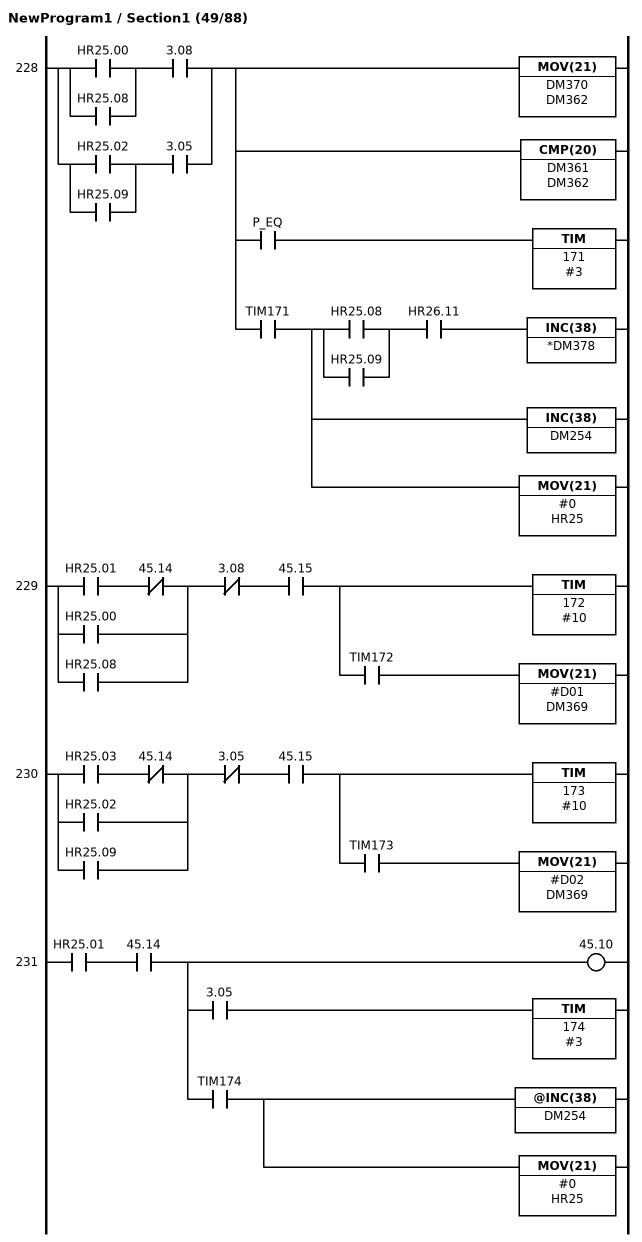
; [picture p48: NewProgram1 / Section1, rungs 228-231]
; rung 228
LD HR25.00
OR HR25.08
AND 3.08
LD HR25.02
OR HR25.09
AND 3.05
ORLD
OUT TR0
MOV(21) DM370 DM362
CMP(20) DM361 DM362
AND P_EQ
TIM 171 #3
LD TR0
AND TIM171
OUT TR0
LD HR25.08
OR HR25.09
ANDLD
AND HR26.11
INC(38) *DM378
LD TR0
INC(38) DM254
MOV(21) #0 HR25
; rung 229
LD HR25.01
ANDNOT 45.14
OR HR25.00
OR HR25.08
ANDNOT 3.08
AND 45.15
TIM 172 #10
AND TIM172
MOV(21) #D01 DM369
; rung 230
LD HR25.03
ANDNOT 45.14
OR HR25.02
OR HR25.09
ANDNOT 3.05
AND 45.15
TIM 173 #10
AND TIM173
MOV(21) #D02 DM369
; rung 231
LD HR25.01
AND 45.14
OUT TR0
OUT 45.10
AND 3.05
TIM 174 #3
LD TR0
AND TIM174
@INC(38) DM254
MOV(21) #0 HR25

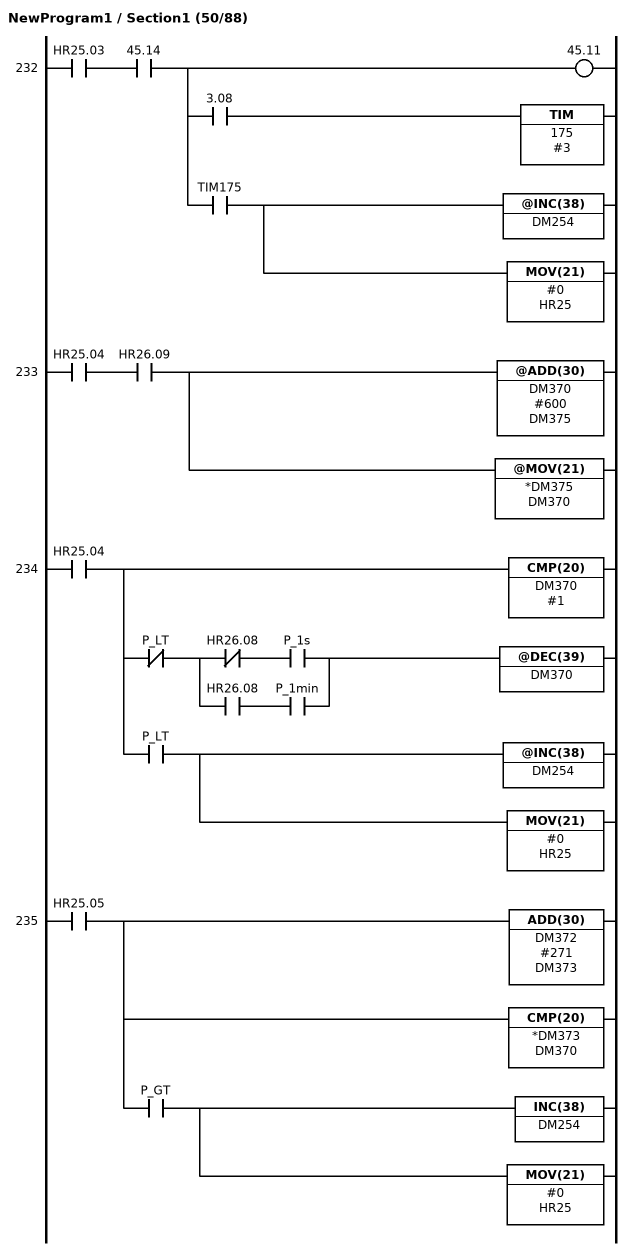
; rung 232
LD HR25.03
AND 45.14
OUT TR0
OUT 45.11
AND 3.08
TIM 175 #3
LD TR0
AND TIM175
@INC(38) DM254
MOV(21) #0 HR25
; rung 233
LD HR25.04
AND HR26.09
@ADD(30) DM370 #600 DM375
@MOV(21) *DM375 DM370
; rung 234
LD HR25.04
OUT TR0
CMP(20) DM370 #1
ANDNOT P_LT
LDNOT HR26.08
AND P_1s
LD HR26.08
AND P_1min
ORLD
ANDLD
@DEC(39) DM370
LD TR0
AND P_LT
@INC(38) DM254
MOV(21) #0 HR25
; rung 235
LD HR25.05
ADD(30) DM372 #271 DM373
CMP(20) *DM373 DM370
AND P_GT
INC(38) DM254
MOV(21) #0 HR25

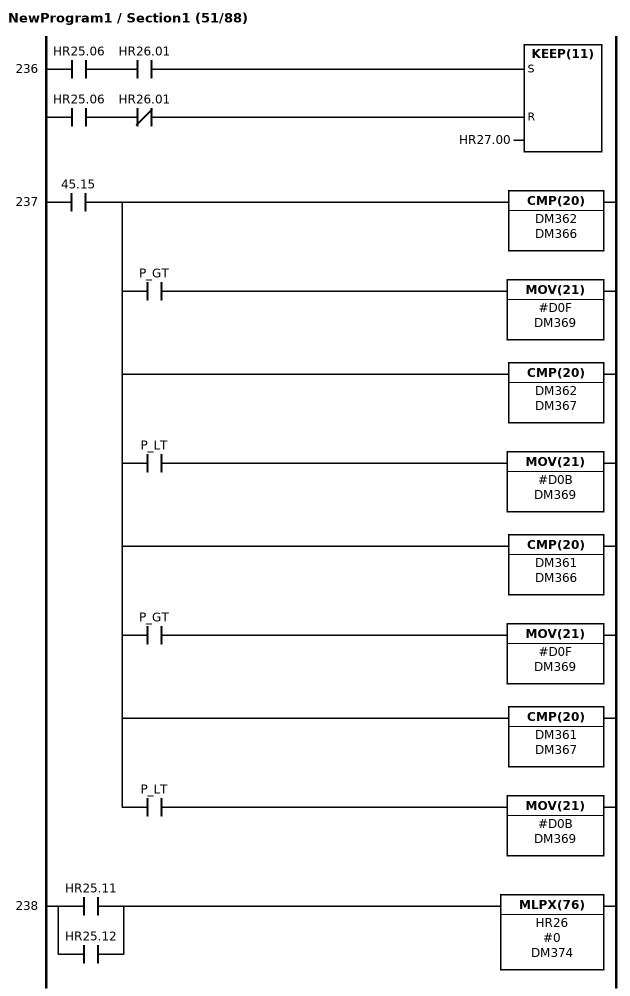
; rung 236
LD HR25.06
AND HR26.01
LD HR25.06
ANDNOT HR26.01
KEEP(11) HR27.00
; rung 237
LD 45.15
OUT TR0
CMP(20) DM362 DM366
AND P_GT
MOV(21) #D0F DM369
LD TR0
CMP(20) DM362 DM367
AND P_LT
MOV(21) #D0B DM369
LD TR0
CMP(20) DM361 DM366
AND P_GT
MOV(21) #D0F DM369
LD TR0
CMP(20) DM361 DM367
AND P_LT
MOV(21) #D0B DM369
; rung 238
LD HR25.11
OR HR25.12
MLPX(76) HR26 #0 DM374

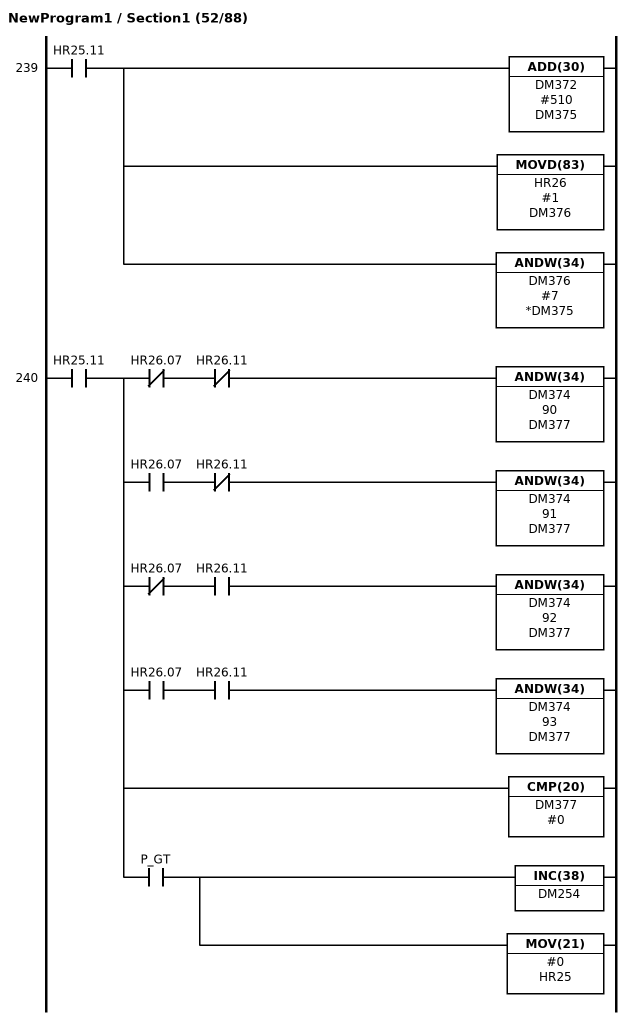
; rung 239
LD HR25.11
ADD(30) DM372 #510 DM375
MOVD(83) HR26 #1 DM376
ANDW(34) DM376 #7 *DM375
; rung 240
LD HR25.11
OUT TR0
ANDNOT HR26.07
ANDNOT HR26.11
ANDW(34) DM374 90 DM377
LD TR0
AND HR26.07
ANDNOT HR26.11
ANDW(34) DM374 91 DM377
LD TR0
ANDNOT HR26.07
AND HR26.11
ANDW(34) DM374 92 DM377
LD TR0
AND HR26.07
AND HR26.11
ANDW(34) DM374 93 DM377
LD TR0
CMP(20) DM377 #0
AND P_GT
INC(38) DM254
MOV(21) #0 HR25

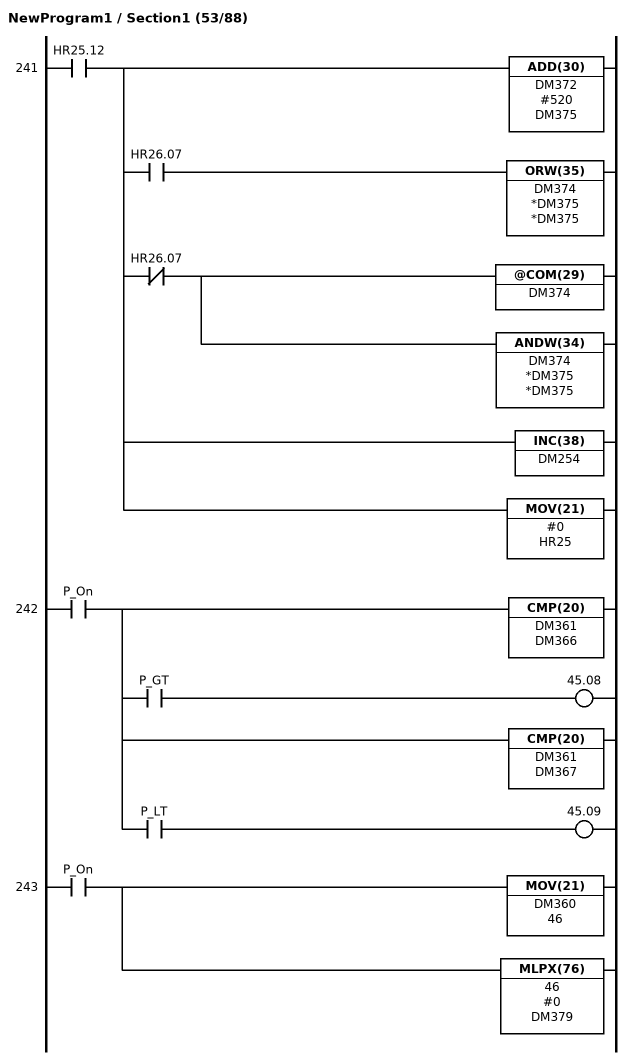
; rung 241
LD HR25.12
OUT TR0
ADD(30) DM372 #520 DM375
AND HR26.07
ORW(35) DM374 *DM375 *DM375
LD TR0
ANDNOT HR26.07
@COM(29) DM374
ANDW(34) DM374 *DM375 *DM375
LD TR0
INC(38) DM254
MOV(21) #0 HR25
; rung 242
LD P_On
OUT TR0
CMP(20) DM361 DM366
AND P_GT
OUT 45.08
LD TR0
CMP(20) DM361 DM367
AND P_LT
OUT 45.09
; rung 243
LD P_On
MOV(21) DM360 46
MLPX(76) 46 #0 DM379

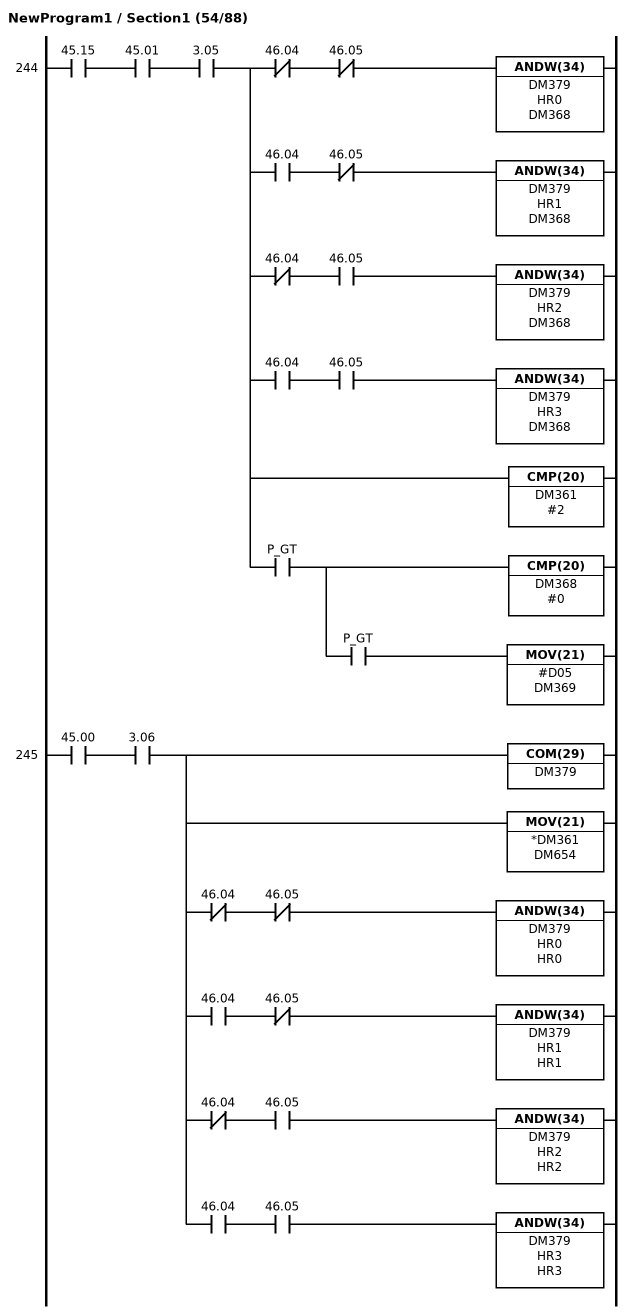
; rung 244
LD 45.15
AND 45.01
AND 3.05
OUT TR0
ANDNOT 46.04
ANDNOT 46.05
ANDW(34) DM379 HR0 DM368
LD TR0
AND 46.04
ANDNOT 46.05
ANDW(34) DM379 HR1 DM368
LD TR0
ANDNOT 46.04
AND 46.05
ANDW(34) DM379 HR2 DM368
LD TR0
AND 46.04
AND 46.05
ANDW(34) DM379 HR3 DM368
LD TR0
CMP(20) DM361 #2
AND P_GT
CMP(20) DM368 #0
AND P_GT
MOV(21) #D05 DM369
; rung 245
LD 45.00
AND 3.06
OUT TR0
COM(29) DM379
MOV(21) *DM361 DM654
ANDNOT 46.04
ANDNOT 46.05
ANDW(34) DM379 HR0 HR0
LD TR0
AND 46.04
ANDNOT 46.05
ANDW(34) DM379 HR1 HR1
LD TR0
ANDNOT 46.04
AND 46.05
ANDW(34) DM379 HR2 HR2
LD TR0
AND 46.04
AND 46.05
ANDW(34) DM379 HR3 HR3

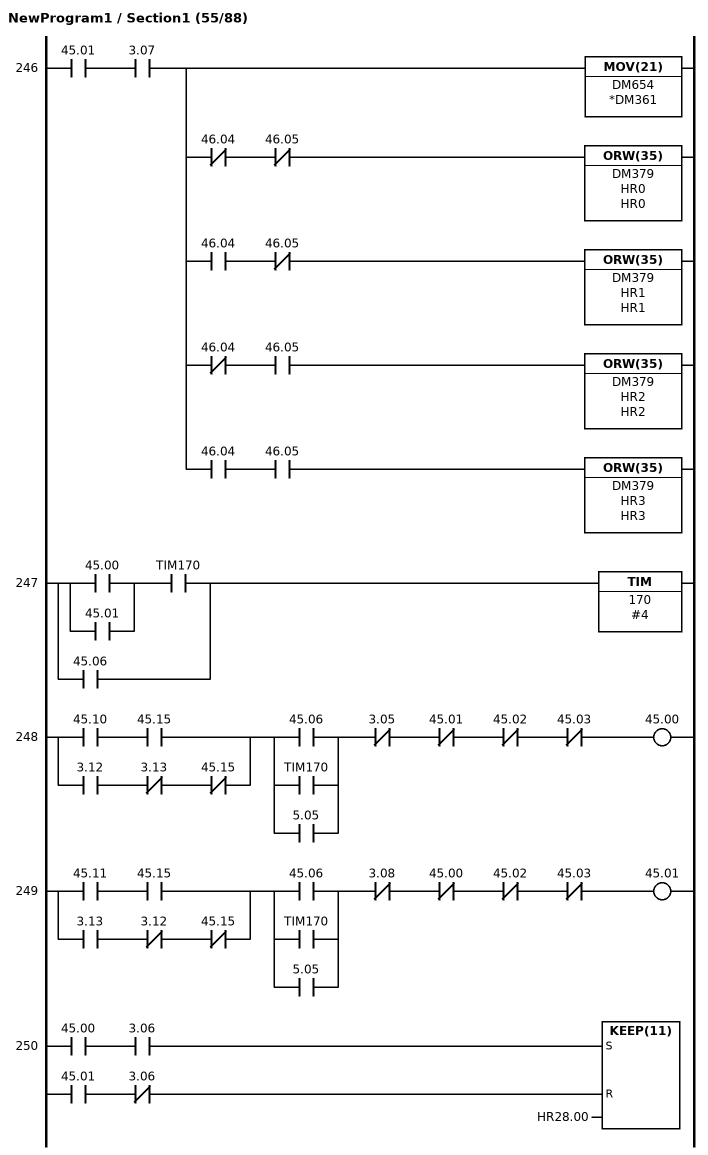
; rung 246
LD 45.01
AND 3.07
OUT TR0
MOV(21) DM654 *DM361
ANDNOT 46.04
ANDNOT 46.05
ORW(35) DM379 HR0 HR0
LD TR0
AND 46.04
ANDNOT 46.05
ORW(35) DM379 HR1 HR1
LD TR0
ANDNOT 46.04
AND 46.05
ORW(35) DM379 HR2 HR2
LD TR0
AND 46.04
AND 46.05
ORW(35) DM379 HR3 HR3
; rung 247
LD 45.00
OR 45.01
AND TIM170
OR 45.06
TIM 170 #4
; rung 248
LD 45.10
AND 45.15
LD 3.12
ANDNOT 3.13
ANDNOT 45.15
ORLD
LD 45.06
OR TIM170
OR 5.05
ANDLD
ANDNOT 3.05
ANDNOT 45.01
ANDNOT 45.02
ANDNOT 45.03
OUT 45.00
; rung 249
LD 45.11
AND 45.15
LD 3.13
ANDNOT 3.12
ANDNOT 45.15
ORLD
LD 45.06
OR TIM170
OR 5.05
ANDLD
ANDNOT 3.08
ANDNOT 45.00
ANDNOT 45.02
ANDNOT 45.03
OUT 45.01
; rung 250
LD 45.00
AND 3.06
LD 45.01
ANDNOT 3.06
KEEP(11) HR28.00

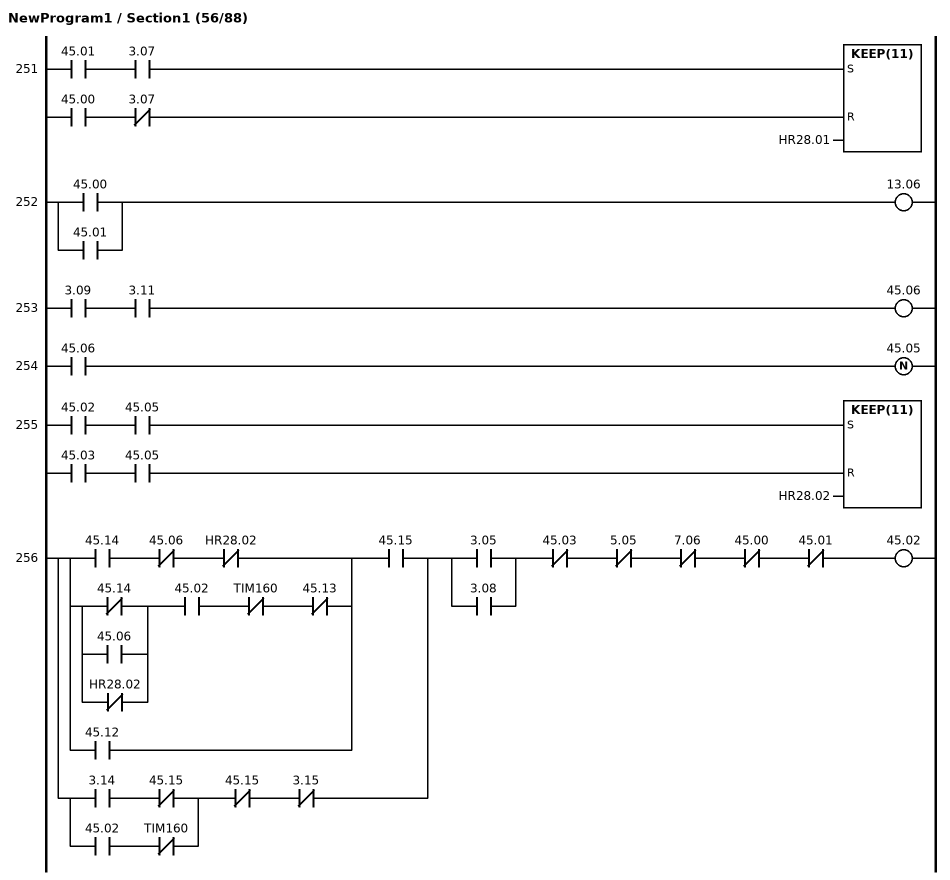
; rung 251
LD 45.01
AND 3.07
LD 45.00
ANDNOT 3.07
KEEP(11) HR28.01
; rung 252
LD 45.00
OR 45.01
OUT 13.06
; rung 253
LD 3.09
AND 3.11
OUT 45.06
; rung 254
LD 45.06
DIFD(14) 45.05
; rung 255
LD 45.02
AND 45.05
LD 45.03
AND 45.05
KEEP(11) HR28.02
; rung 256
LD 45.14
ANDNOT 45.06
ANDNOT HR28.02
LDNOT 45.14
OR 45.06
ORNOT HR28.02
AND 45.02
ANDNOT TIM160
ANDNOT 45.13
ORLD
OR 45.12
AND 45.15
LD 3.14
ANDNOT 45.15
LD 45.02
ANDNOT TIM160
ORLD
ANDNOT 45.15
ANDNOT 3.15
ORLD
LD 3.05
OR 3.08
ANDLD
ANDNOT 45.03
ANDNOT 5.05
ANDNOT 7.06
ANDNOT 45.00
ANDNOT 45.01
OUT 45.02

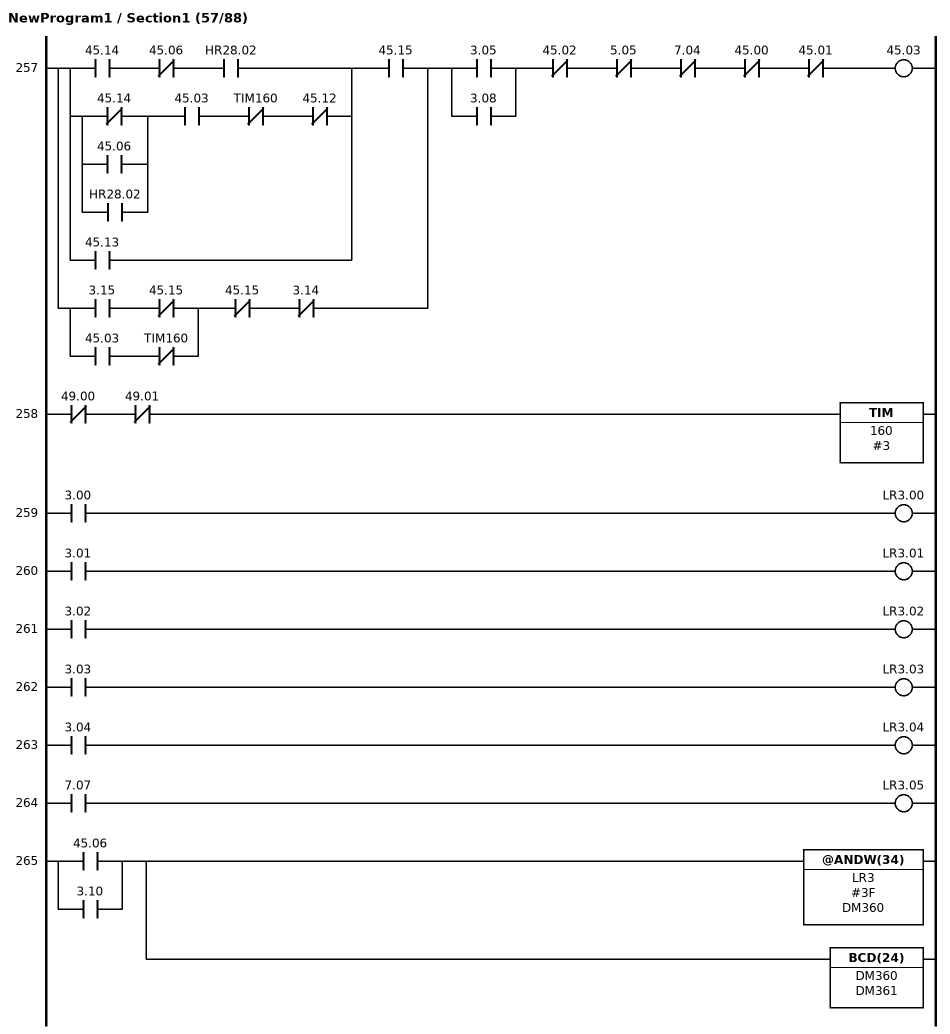
; rung 257
LD 45.14
ANDNOT 45.06
AND HR28.02
LDNOT 45.14
OR 45.06
OR HR28.02
AND 45.03
ANDNOT TIM160
ANDNOT 45.12
ORLD
OR 45.13
AND 45.15
LD 3.15
ANDNOT 45.15
LD 45.03
ANDNOT TIM160
ORLD
ANDNOT 45.15
ANDNOT 3.14
ORLD
LD 3.05
OR 3.08
ANDLD
ANDNOT 45.02
ANDNOT 5.05
ANDNOT 7.04
ANDNOT 45.00
ANDNOT 45.01
OUT 45.03
; rung 258
LDNOT 49.00
ANDNOT 49.01
TIM 160 #3
; rung 259
LD 3.00
OUT LR3.00
; rung 260
LD 3.01
OUT LR3.01
; rung 261
LD 3.02
OUT LR3.02
; rung 262
LD 3.03
OUT LR3.03
; rung 263
LD 3.04
OUT LR3.04
; rung 264
LD 7.07
OUT LR3.05
; rung 265
LD 45.06
OR 3.10
@ANDW(34) LR3 #3F DM360
BCD(24) DM360 DM361

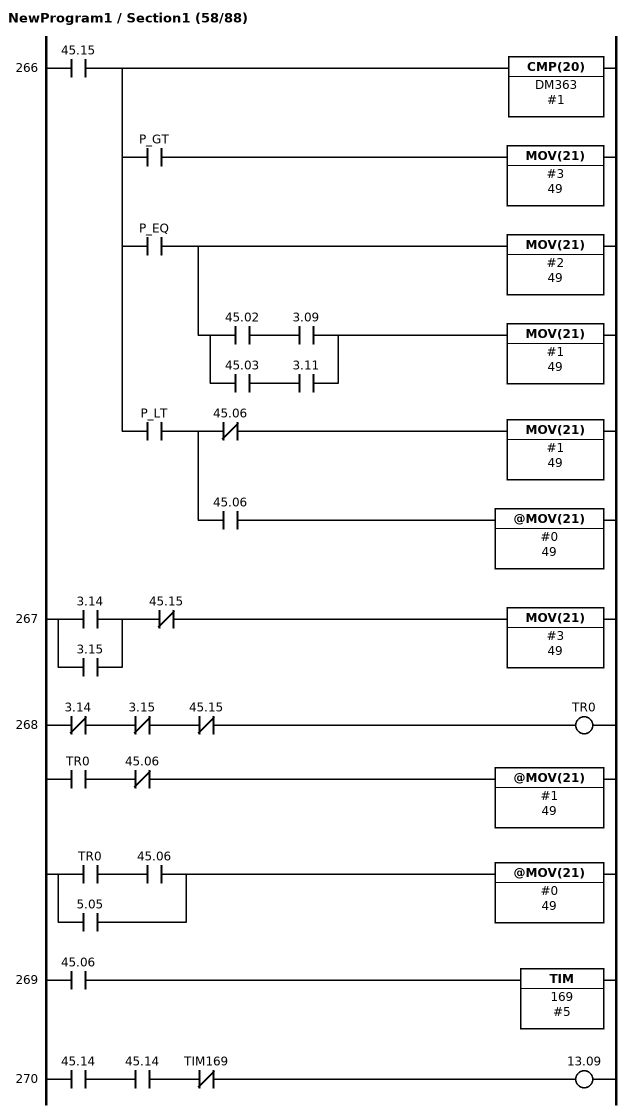
; rung 266
LD 45.15
OUT TR0
CMP(20) DM363 #1
AND P_GT
MOV(21) #3 49
LD TR0
AND P_EQ
MOV(21) #2 49
LD 45.02
AND 3.09
LD 45.03
AND 3.11
ORLD
ANDLD
MOV(21) #1 49
LD TR0
AND P_LT
OUT TR0
ANDNOT 45.06
MOV(21) #1 49
LD TR0
AND 45.06
@MOV(21) #0 49
; rung 267
LD 3.14
OR 3.15
ANDNOT 45.15
MOV(21) #3 49
; rung 268
LDNOT 3.14
ANDNOT 3.15
ANDNOT 45.15
OUT TR0
ANDNOT 45.06
@MOV(21) #1 49
LD TR0
AND 45.06
OR 5.05
@MOV(21) #0 49
; rung 269
LD 45.06
TIM 169 #5
; rung 270
LD 45.14
AND 45.14
ANDNOT TIM169
OUT 13.09

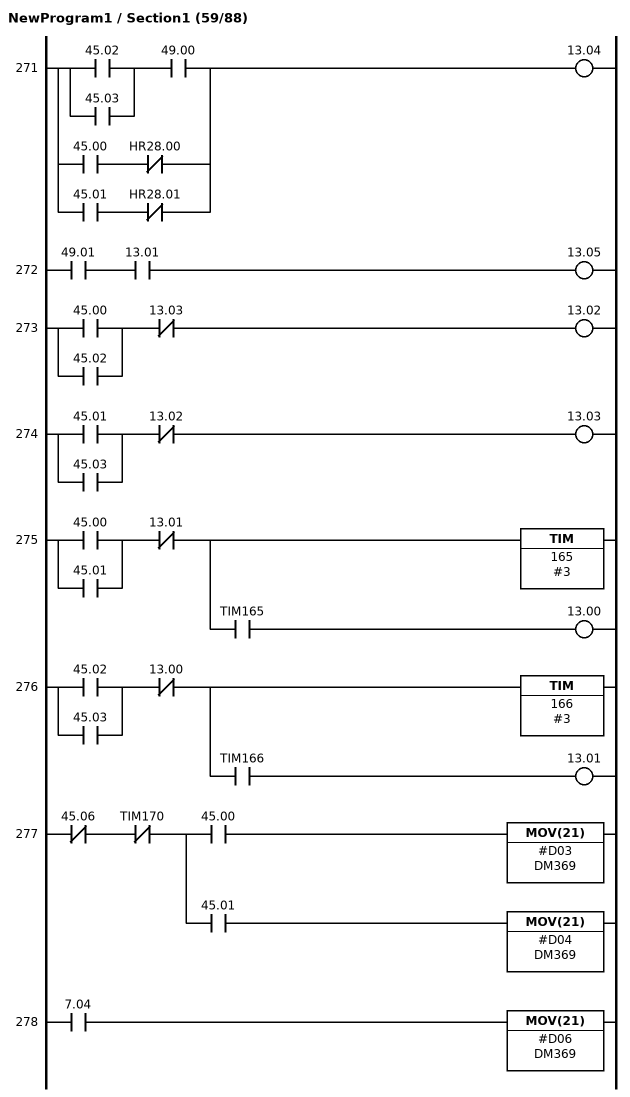
; rung 271
LD 45.02
OR 45.03
AND 49.00
LD 45.00
ANDNOT HR28.00
ORLD
LD 45.01
ANDNOT HR28.01
ORLD
OUT 13.04
; rung 272
LD 49.01
AND 13.01
OUT 13.05
; rung 273
LD 45.00
OR 45.02
ANDNOT 13.03
OUT 13.02
; rung 274
LD 45.01
OR 45.03
ANDNOT 13.02
OUT 13.03
; rung 275
LD 45.00
OR 45.01
ANDNOT 13.01
TIM 165 #3
AND TIM165
OUT 13.00
; rung 276
LD 45.02
OR 45.03
ANDNOT 13.00
TIM 166 #3
AND TIM166
OUT 13.01
; rung 277
LDNOT 45.06
ANDNOT TIM170
OUT TR0
AND 45.00
MOV(21) #D03 DM369
LD TR0
AND 45.01
MOV(21) #D04 DM369
; rung 278
LD 7.04
MOV(21) #D06 DM369

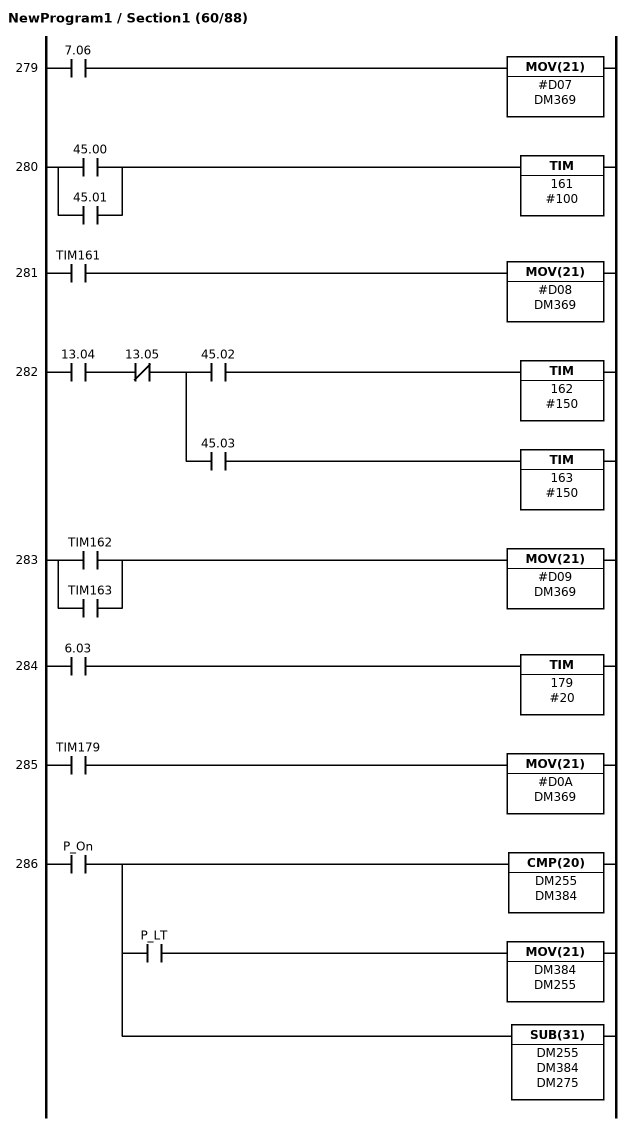
; rung 279
LD 7.06
MOV(21) #D07 DM369
; rung 280
LD 45.00
OR 45.01
TIM 161 #100
; rung 281
LD TIM161
MOV(21) #D08 DM369
; rung 282
LD 13.04
ANDNOT 13.05
OUT TR0
AND 45.02
TIM 162 #150
LD TR0
AND 45.03
TIM 163 #150
; rung 283
LD TIM162
OR TIM163
MOV(21) #D09 DM369
; rung 284
LD 6.03
TIM 179 #20
; rung 285
LD TIM179
MOV(21) #D0A DM369
; rung 286
LD P_On
OUT TR0
CMP(20) DM255 DM384
AND P_LT
MOV(21) DM384 DM255
LD TR0
SUB(31) DM255 DM384 DM275

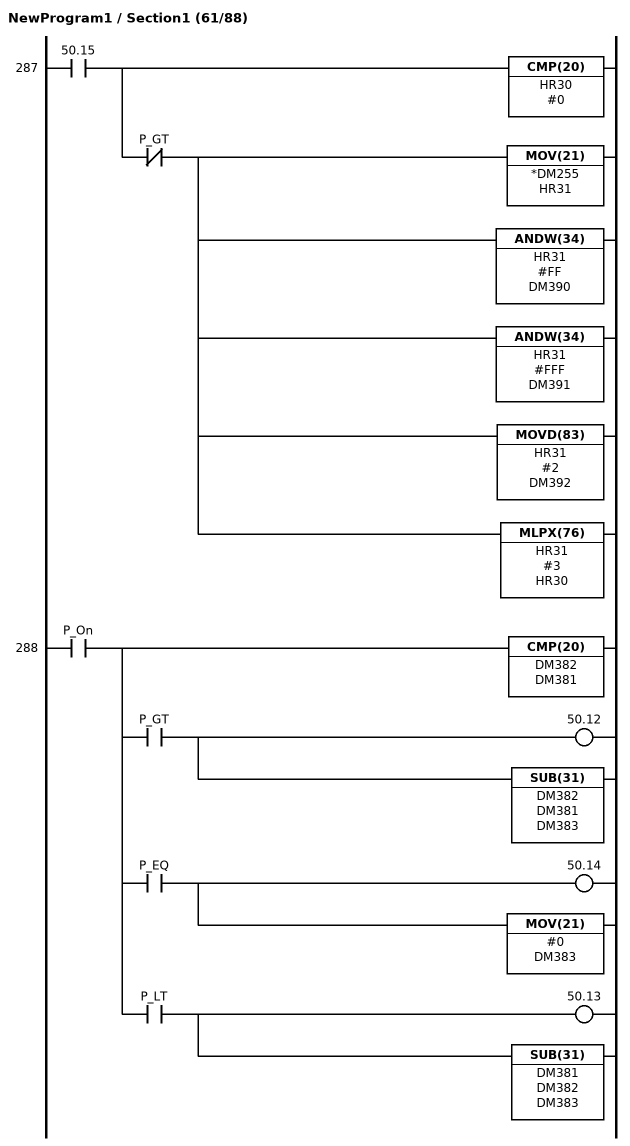
; rung 287
LD 50.15
CMP(20) HR30 #0
ANDNOT P_GT
MOV(21) *DM255 HR31
ANDW(34) HR31 #FF DM390
ANDW(34) HR31 #FFF DM391
MOVD(83) HR31 #2 DM392
MLPX(76) HR31 #3 HR30
; rung 288
LD P_On
OUT TR0
CMP(20) DM382 DM381
AND P_GT
OUT 50.12
SUB(31) DM382 DM381 DM383
LD TR0
AND P_EQ
OUT 50.14
MOV(21) #0 DM383
LD TR0
AND P_LT
OUT 50.13
SUB(31) DM381 DM382 DM383

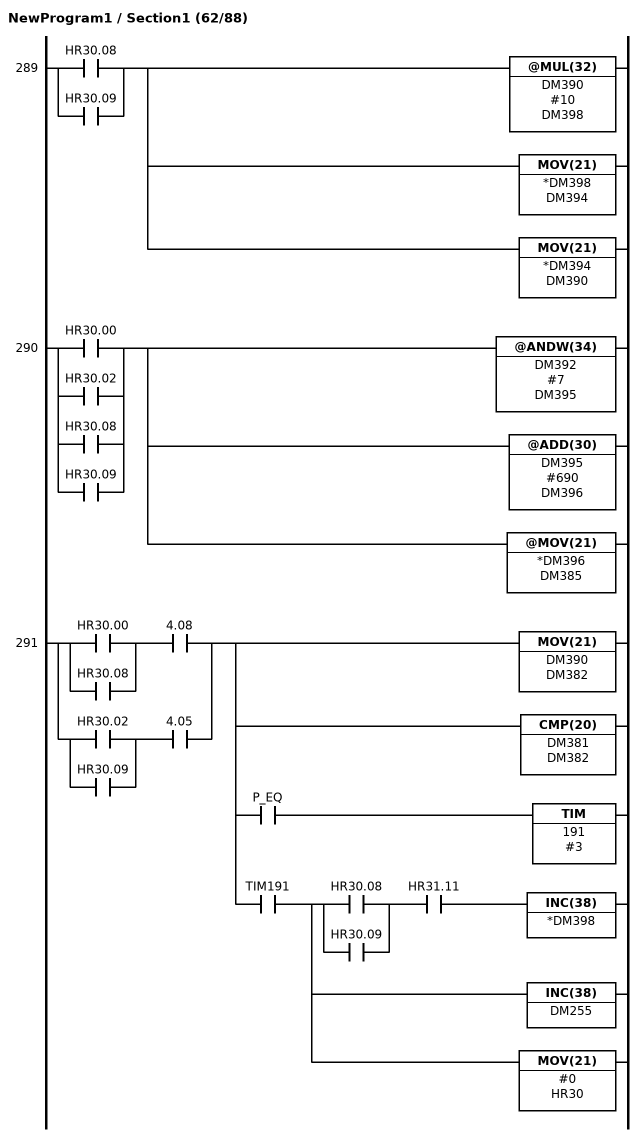
; rung 289
LD HR30.08
OR HR30.09
@MUL(32) DM390 #10 DM398
MOV(21) *DM398 DM394
MOV(21) *DM394 DM390
; rung 290
LD HR30.00
OR HR30.02
OR HR30.08
OR HR30.09
@ANDW(34) DM392 #7 DM395
@ADD(30) DM395 #690 DM396
@MOV(21) *DM396 DM385
; rung 291
LD HR30.00
OR HR30.08
AND 4.08
LD HR30.02
OR HR30.09
AND 4.05
ORLD
OUT TR0
MOV(21) DM390 DM382
CMP(20) DM381 DM382
AND P_EQ
TIM 191 #3
LD TR0
AND TIM191
OUT TR0
LD HR30.08
OR HR30.09
ANDLD
AND HR31.11
INC(38) *DM398
LD TR0
INC(38) DM255
MOV(21) #0 HR30

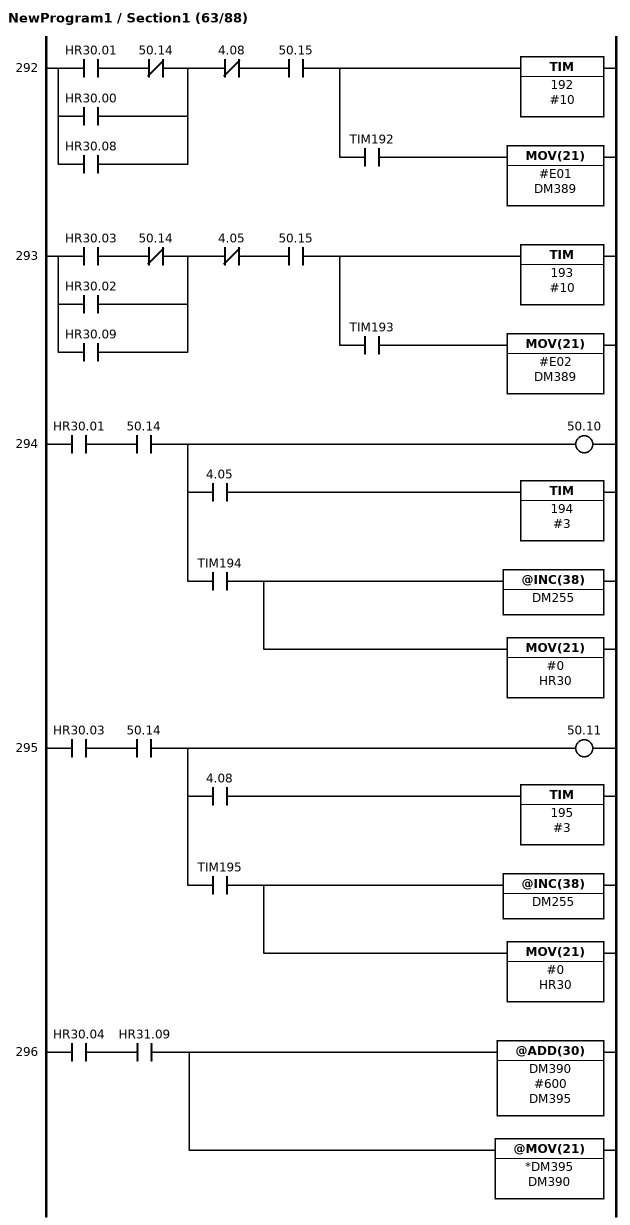
; rung 292
LD HR30.01
ANDNOT 50.14
OR HR30.00
OR HR30.08
ANDNOT 4.08
AND 50.15
TIM 192 #10
AND TIM192
MOV(21) #E01 DM389
; rung 293
LD HR30.03
ANDNOT 50.14
OR HR30.02
OR HR30.09
ANDNOT 4.05
AND 50.15
TIM 193 #10
AND TIM193
MOV(21) #E02 DM389
; rung 294
LD HR30.01
AND 50.14
OUT TR0
OUT 50.10
AND 4.05
TIM 194 #3
LD TR0
AND TIM194
@INC(38) DM255
MOV(21) #0 HR30
; rung 295
LD HR30.03
AND 50.14
OUT TR0
OUT 50.11
AND 4.08
TIM 195 #3
LD TR0
AND TIM195
@INC(38) DM255
MOV(21) #0 HR30
; rung 296
LD HR30.04
AND HR31.09
@ADD(30) DM390 #600 DM395
@MOV(21) *DM395 DM390

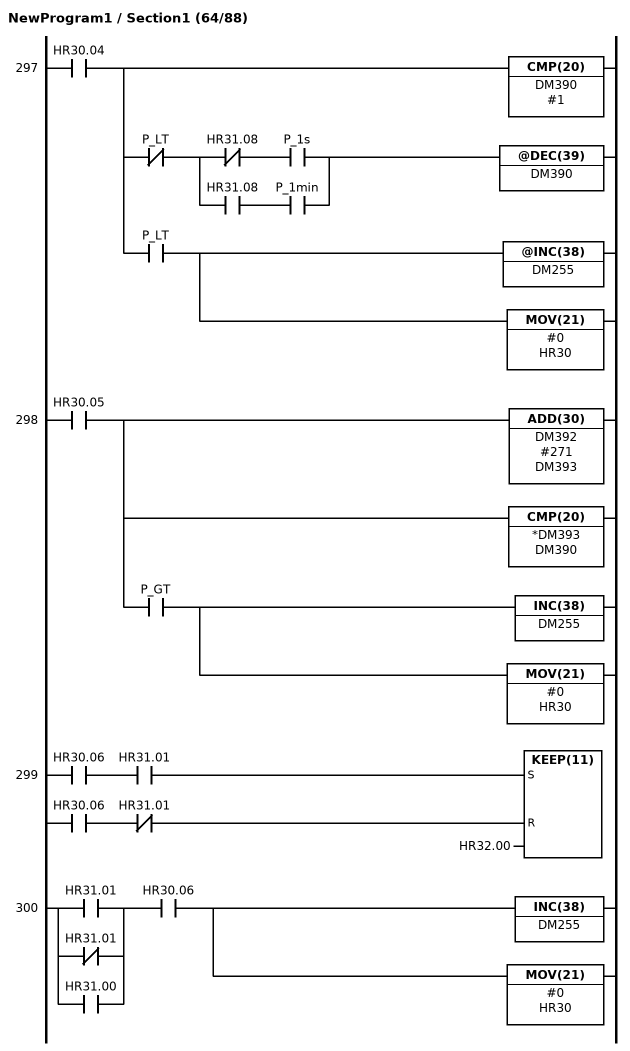
; rung 297
LD HR30.04
OUT TR0
CMP(20) DM390 #1
ANDNOT P_LT
LDNOT HR31.08
AND P_1s
LD HR31.08
AND P_1min
ORLD
ANDLD
@DEC(39) DM390
LD TR0
AND P_LT
@INC(38) DM255
MOV(21) #0 HR30
; rung 298
LD HR30.05
ADD(30) DM392 #271 DM393
CMP(20) *DM393 DM390
AND P_GT
INC(38) DM255
MOV(21) #0 HR30
; rung 299
LD HR30.06
AND HR31.01
LD HR30.06
ANDNOT HR31.01
KEEP(11) HR32.00
; rung 300
LD HR31.01
ORNOT HR31.01
OR HR31.00
AND HR30.06
INC(38) DM255
MOV(21) #0 HR30

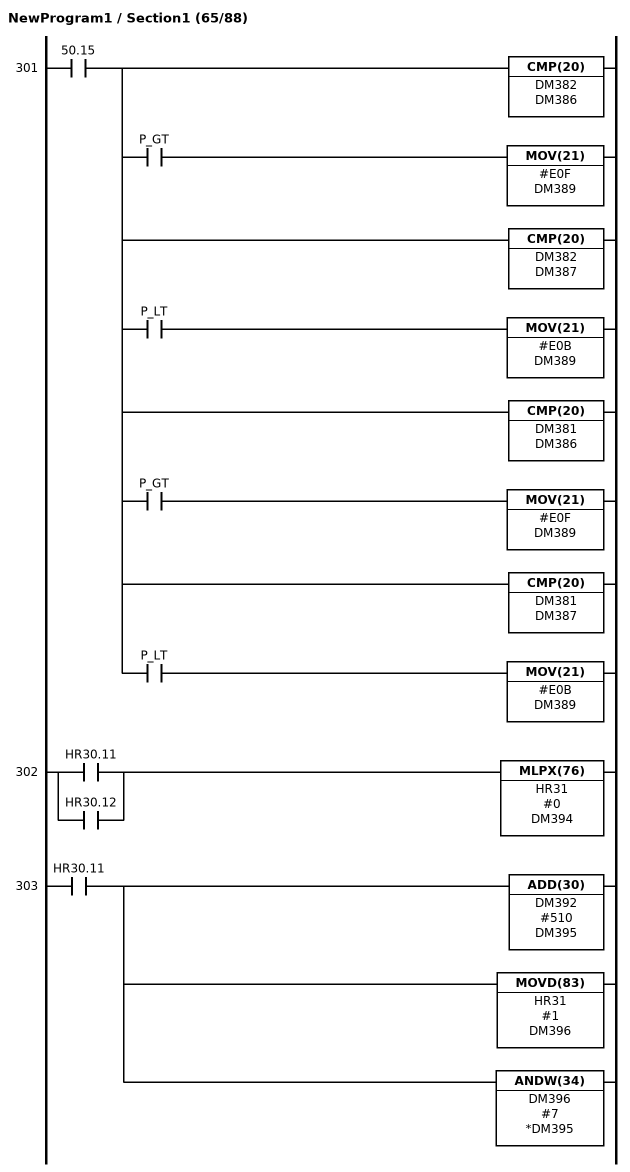
; rung 301
LD 50.15
OUT TR0
CMP(20) DM382 DM386
AND P_GT
MOV(21) #E0F DM389
LD TR0
CMP(20) DM382 DM387
AND P_LT
MOV(21) #E0B DM389
LD TR0
CMP(20) DM381 DM386
AND P_GT
MOV(21) #E0F DM389
LD TR0
CMP(20) DM381 DM387
AND P_LT
MOV(21) #E0B DM389
; rung 302
LD HR30.11
OR HR30.12
MLPX(76) HR31 #0 DM394
; rung 303
LD HR30.11
ADD(30) DM392 #510 DM395
MOVD(83) HR31 #1 DM396
ANDW(34) DM396 #7 *DM395

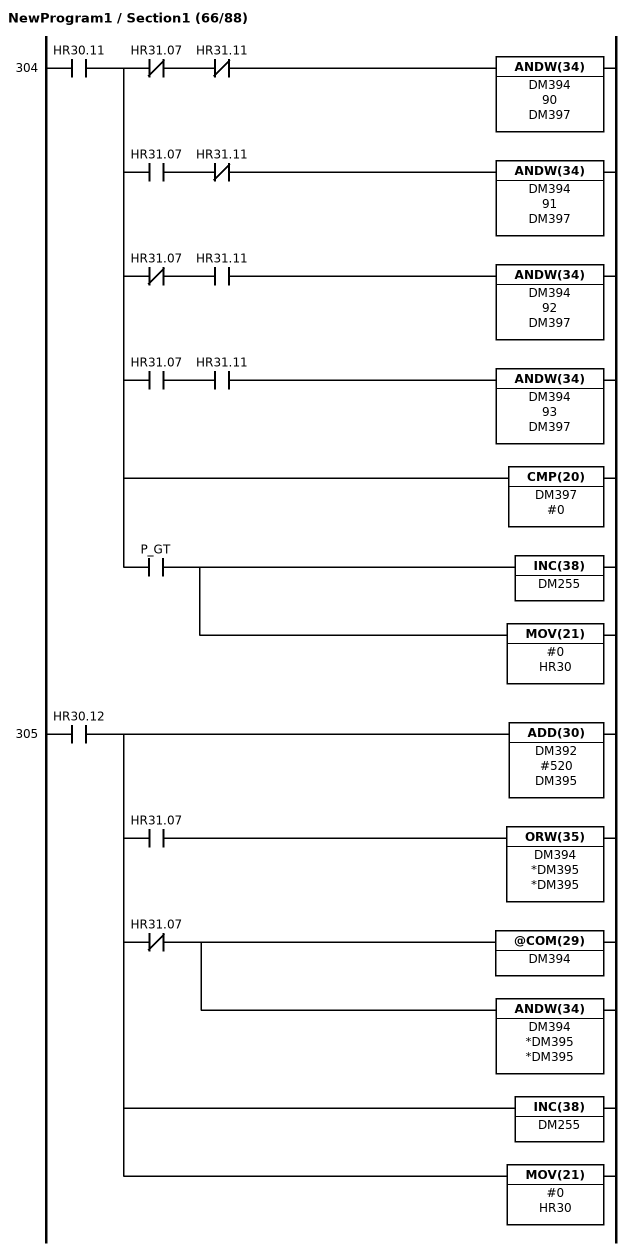
; rung 304
LD HR30.11
OUT TR0
ANDNOT HR31.07
ANDNOT HR31.11
ANDW(34) DM394 90 DM397
LD TR0
AND HR31.07
ANDNOT HR31.11
ANDW(34) DM394 91 DM397
LD TR0
ANDNOT HR31.07
AND HR31.11
ANDW(34) DM394 92 DM397
LD TR0
AND HR31.07
AND HR31.11
ANDW(34) DM394 93 DM397
LD TR0
CMP(20) DM397 #0
AND P_GT
INC(38) DM255
MOV(21) #0 HR30
; rung 305
LD HR30.12
OUT TR0
ADD(30) DM392 #520 DM395
AND HR31.07
ORW(35) DM394 *DM395 *DM395
LD TR0
ANDNOT HR31.07
@COM(29) DM394
ANDW(34) DM394 *DM395 *DM395
LD TR0
INC(38) DM255
MOV(21) #0 HR30

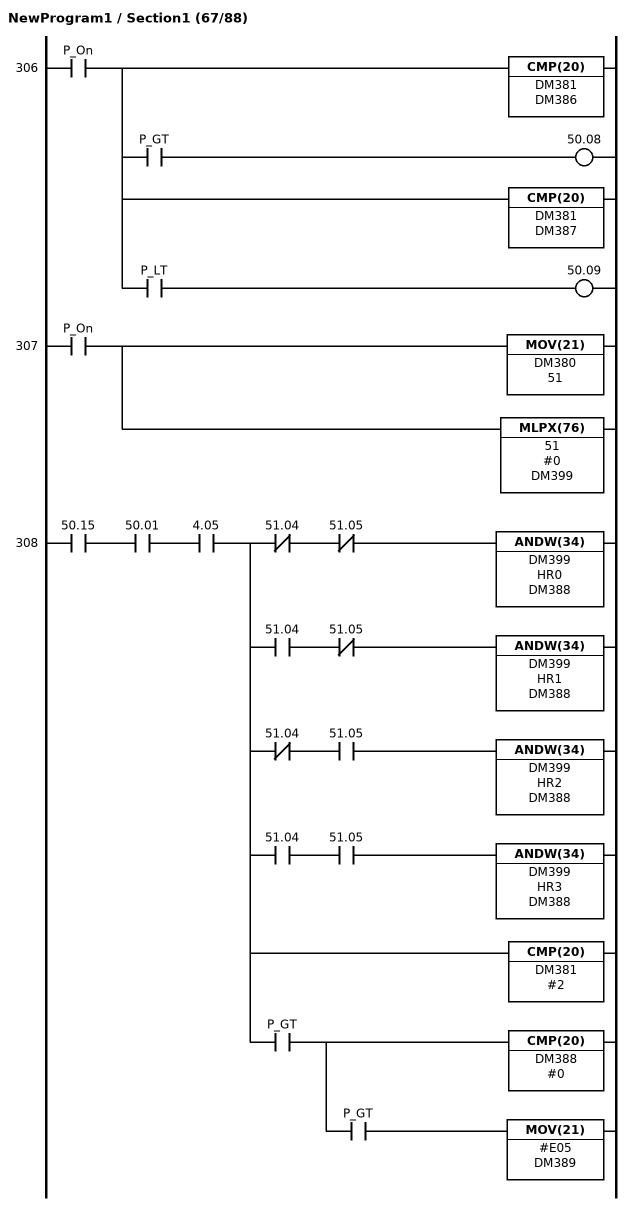
; rung 306
LD P_On
OUT TR0
CMP(20) DM381 DM386
AND P_GT
OUT 50.08
LD TR0
CMP(20) DM381 DM387
AND P_LT
OUT 50.09
; rung 307
LD P_On
MOV(21) DM380 51
MLPX(76) 51 #0 DM399
; rung 308
LD 50.15
AND 50.01
AND 4.05
OUT TR0
ANDNOT 51.04
ANDNOT 51.05
ANDW(34) DM399 HR0 DM388
LD TR0
AND 51.04
ANDNOT 51.05
ANDW(34) DM399 HR1 DM388
LD TR0
ANDNOT 51.04
AND 51.05
ANDW(34) DM399 HR2 DM388
LD TR0
AND 51.04
AND 51.05
ANDW(34) DM399 HR3 DM388
LD TR0
CMP(20) DM381 #2
AND P_GT
CMP(20) DM388 #0
AND P_GT
MOV(21) #E05 DM389

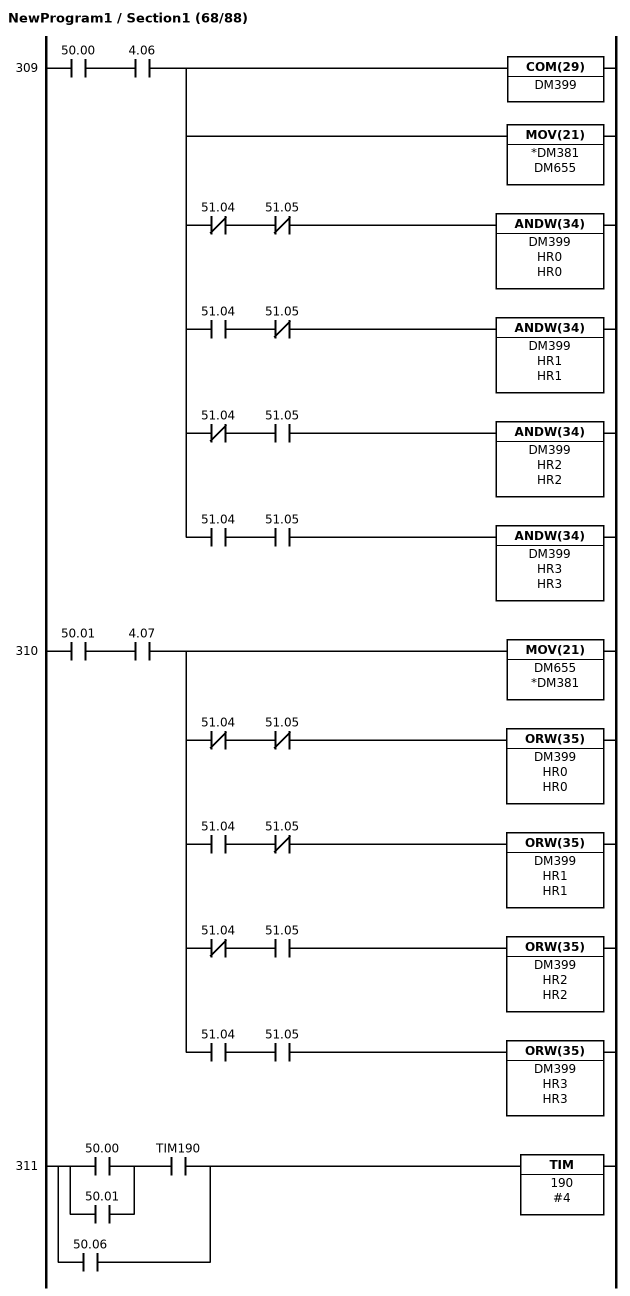
; rung 309
LD 50.00
AND 4.06
OUT TR0
COM(29) DM399
MOV(21) *DM381 DM655
ANDNOT 51.04
ANDNOT 51.05
ANDW(34) DM399 HR0 HR0
LD TR0
AND 51.04
ANDNOT 51.05
ANDW(34) DM399 HR1 HR1
LD TR0
ANDNOT 51.04
AND 51.05
ANDW(34) DM399 HR2 HR2
LD TR0
AND 51.04
AND 51.05
ANDW(34) DM399 HR3 HR3
; rung 310
LD 50.01
AND 4.07
OUT TR0
MOV(21) DM655 *DM381
ANDNOT 51.04
ANDNOT 51.05
ORW(35) DM399 HR0 HR0
LD TR0
AND 51.04
ANDNOT 51.05
ORW(35) DM399 HR1 HR1
LD TR0
ANDNOT 51.04
AND 51.05
ORW(35) DM399 HR2 HR2
LD TR0
AND 51.04
AND 51.05
ORW(35) DM399 HR3 HR3
; rung 311
LD 50.00
OR 50.01
AND TIM190
OR 50.06
TIM 190 #4

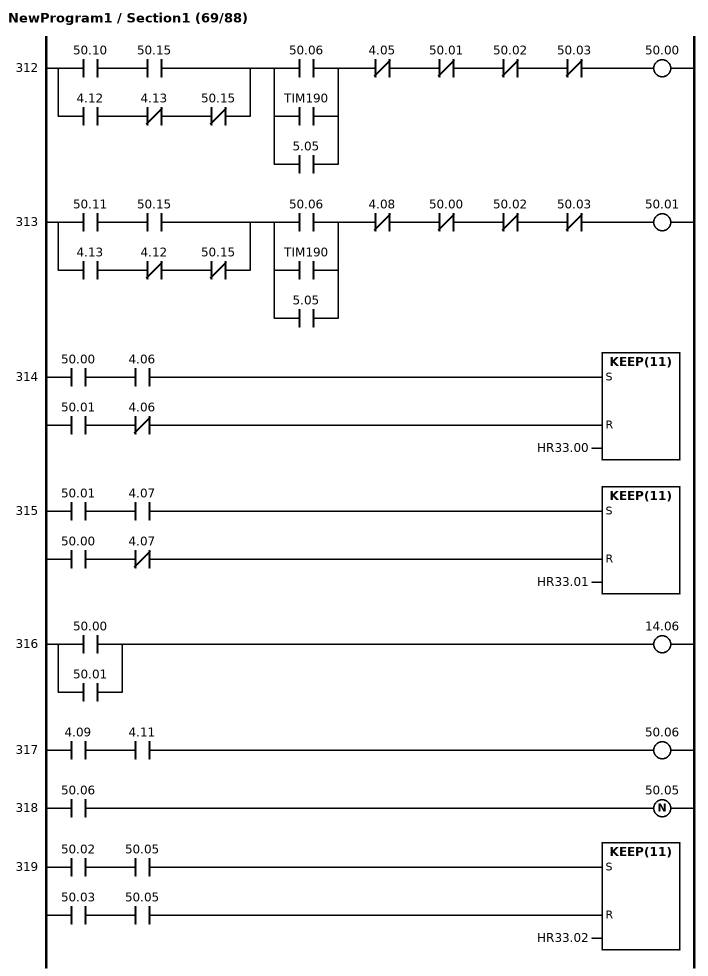
; rung 312
LD 50.10
AND 50.15
LD 4.12
ANDNOT 4.13
ANDNOT 50.15
ORLD
LD 50.06
OR TIM190
OR 5.05
ANDLD
ANDNOT 4.05
ANDNOT 50.01
ANDNOT 50.02
ANDNOT 50.03
OUT 50.00
; rung 313
LD 50.11
AND 50.15
LD 4.13
ANDNOT 4.12
ANDNOT 50.15
ORLD
LD 50.06
OR TIM190
OR 5.05
ANDLD
ANDNOT 4.08
ANDNOT 50.00
ANDNOT 50.02
ANDNOT 50.03
OUT 50.01
; rung 314
LD 50.00
AND 4.06
LD 50.01
ANDNOT 4.06
KEEP(11) HR33.00
; rung 315
LD 50.01
AND 4.07
LD 50.00
ANDNOT 4.07
KEEP(11) HR33.01
; rung 316
LD 50.00
OR 50.01
OUT 14.06
; rung 317
LD 4.09
AND 4.11
OUT 50.06
; rung 318
LD 50.06
DIFD(14) 50.05
; rung 319
LD 50.02
AND 50.05
LD 50.03
AND 50.05
KEEP(11) HR33.02

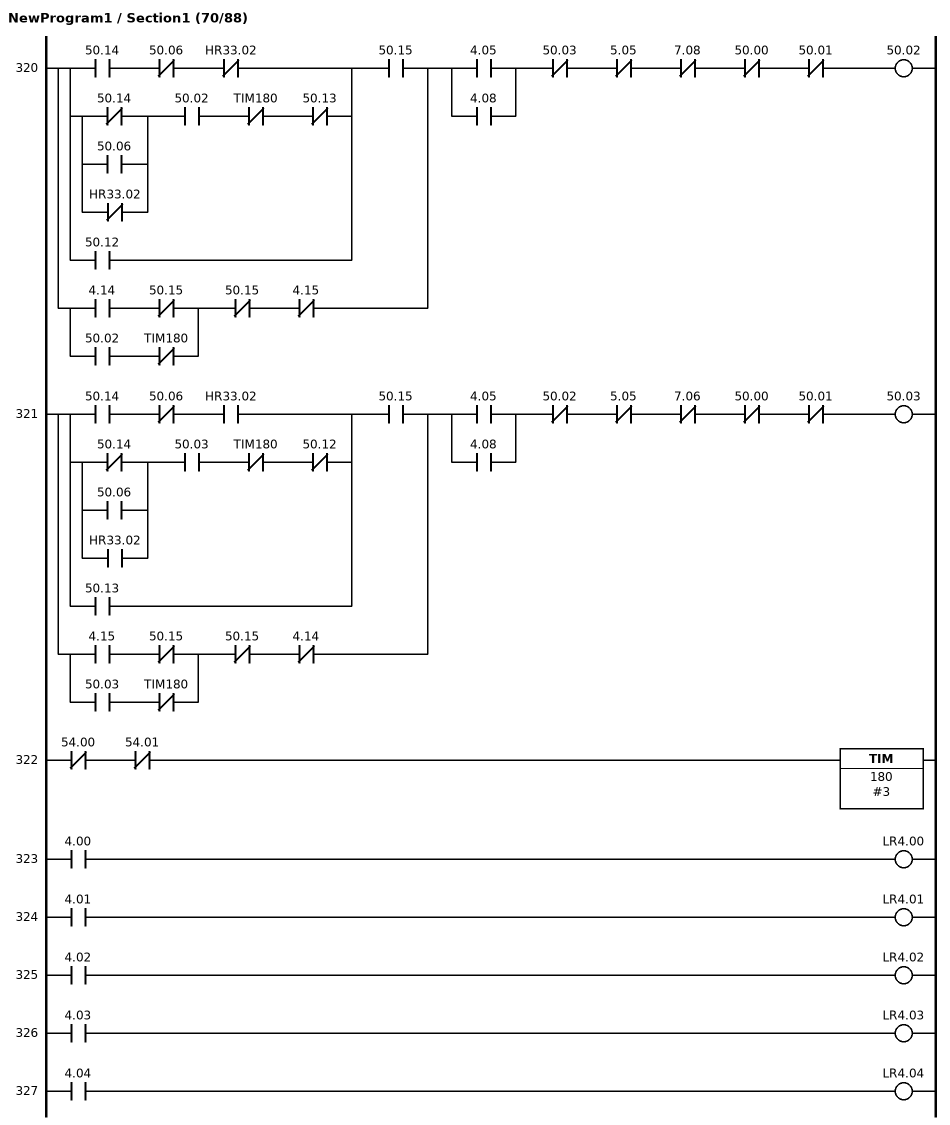
; rung 320
LD 50.14
ANDNOT 50.06
ANDNOT HR33.02
LDNOT 50.14
OR 50.06
ORNOT HR33.02
AND 50.02
ANDNOT TIM180
ANDNOT 50.13
ORLD
OR 50.12
AND 50.15
LD 4.14
ANDNOT 50.15
LD 50.02
ANDNOT TIM180
ORLD
ANDNOT 50.15
ANDNOT 4.15
ORLD
LD 4.05
OR 4.08
ANDLD
ANDNOT 50.03
ANDNOT 5.05
ANDNOT 7.08
ANDNOT 50.00
ANDNOT 50.01
OUT 50.02
; rung 321
LD 50.14
ANDNOT 50.06
AND HR33.02
LDNOT 50.14
OR 50.06
OR HR33.02
AND 50.03
ANDNOT TIM180
ANDNOT 50.12
ORLD
OR 50.13
AND 50.15
LD 4.15
ANDNOT 50.15
LD 50.03
ANDNOT TIM180
ORLD
ANDNOT 50.15
ANDNOT 4.14
ORLD
LD 4.05
OR 4.08
ANDLD
ANDNOT 50.02
ANDNOT 5.05
ANDNOT 7.06
ANDNOT 50.00
ANDNOT 50.01
OUT 50.03
; rung 322
LDNOT 54.00
ANDNOT 54.01
TIM 180 #3
; rung 323
LD 4.00
OUT LR4.00
; rung 324
LD 4.01
OUT LR4.01
; rung 325
LD 4.02
OUT LR4.02
; rung 326
LD 4.03
OUT LR4.03
; rung 327
LD 4.04
OUT LR4.04

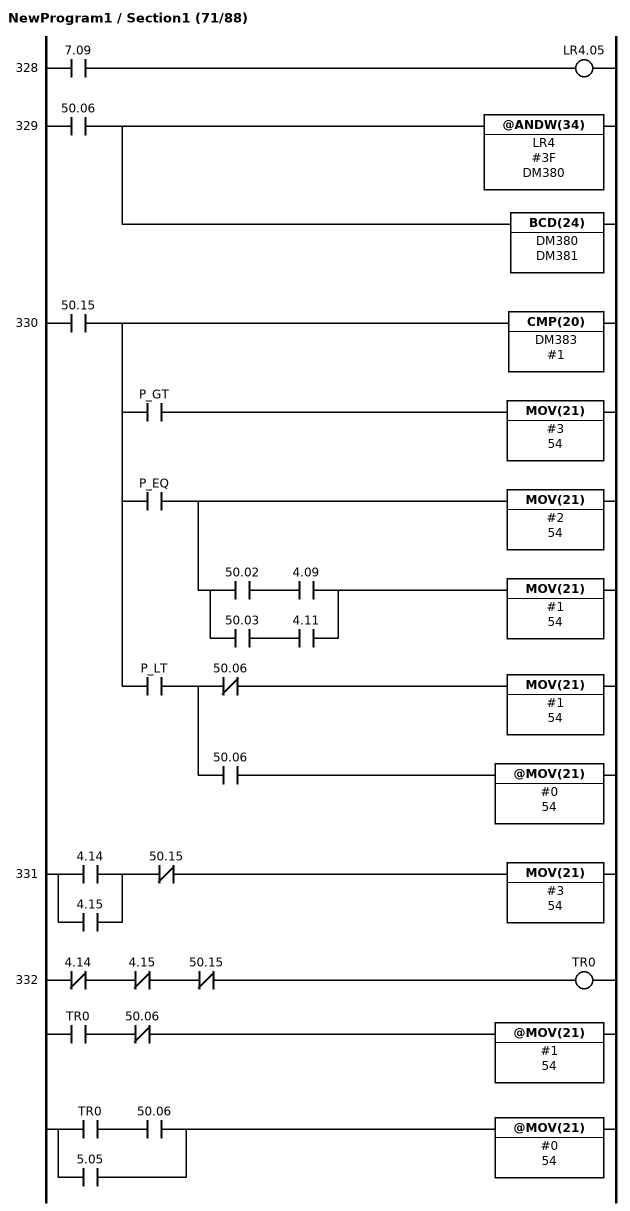
; rung 328
LD 7.09
OUT LR4.05
; rung 329
LD 50.06
@ANDW(34) LR4 #3F DM380
BCD(24) DM380 DM381
; rung 330
LD 50.15
OUT TR0
CMP(20) DM383 #1
AND P_GT
MOV(21) #3 54
LD TR0
AND P_EQ
MOV(21) #2 54
LD 50.02
AND 4.09
LD 50.03
AND 4.11
ORLD
ANDLD
MOV(21) #1 54
LD TR0
AND P_LT
OUT TR0
ANDNOT 50.06
MOV(21) #1 54
LD TR0
AND 50.06
@MOV(21) #0 54
; rung 331
LD 4.14
OR 4.15
ANDNOT 50.15
MOV(21) #3 54
; rung 332
LDNOT 4.14
ANDNOT 4.15
ANDNOT 50.15
OUT TR0
ANDNOT 50.06
@MOV(21) #1 54
LD TR0
AND 50.06
OR 5.05
@MOV(21) #0 54

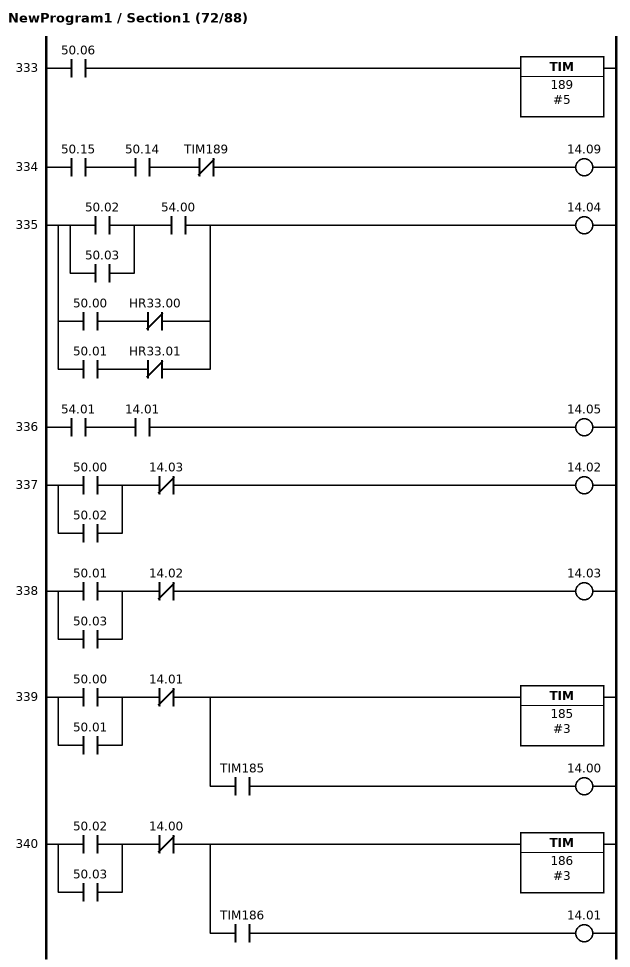
; rung 333
LD 50.06
TIM 189 #5
; rung 334
LD 50.15
AND 50.14
ANDNOT TIM189
OUT 14.09
; rung 335
LD 50.02
OR 50.03
AND 54.00
LD 50.00
ANDNOT HR33.00
ORLD
LD 50.01
ANDNOT HR33.01
ORLD
OUT 14.04
; rung 336
LD 54.01
AND 14.01
OUT 14.05
; rung 337
LD 50.00
OR 50.02
ANDNOT 14.03
OUT 14.02
; rung 338
LD 50.01
OR 50.03
ANDNOT 14.02
OUT 14.03
; rung 339
LD 50.00
OR 50.01
ANDNOT 14.01
TIM 185 #3
AND TIM185
OUT 14.00
; rung 340
LD 50.02
OR 50.03
ANDNOT 14.00
TIM 186 #3
AND TIM186
OUT 14.01

